Yaskawa INFORM job: ID_TEST.JBI

/JOB
//NAME ID_TEST
///FOLDERNAME TWINCAT_KOMMUNIKATION
//POS
///NPOS 0,0,0,0,0,0
//INST
///DATE 2020/06/10 10:42
///ATTR SC,RW
NOP
'SET_ID
CALL JOB:SET_ID ARGF111 ARGF"WID"
TIMER T=1.00
CALL JOB:SET_ID ARGF222 ARGF"NAHT_NR"
TIMER T=1.00
CALL JOB:SET_ID ARGF333 ARGF"LAGE_NR"
TIMER T=1.00
CALL JOB:SET_ID ARGF444 ARGF"RAUPE_NR"
TIMER T=1.00
'GET_ID
CALL JOB:GET_ID ARGF"WID"
TIMER T=1.00
CALL JOB:GET_ID ARGF"NAHT_NR"
TIMER T=1.00
CALL JOB:GET_ID ARGF"LAGE_NR"
TIMER T=1.00
CALL JOB:GET_ID ARGF"RAUPE_NR"
TIMER T=1.00
CALL JOB:SET_ID_MANUEL
END
